KUKA KRL program: CNCRMsgs.src, CNCRMsgs.dat

--- CNCRMsgs.src ---
&ACCESS RV
&REL 50
&PARAM EDITMASK = *
&PARAM TEMPLATE = C:\KRC\Roboter\Template\ExpertVorgabe
DEF CNCRMsgs( )

;************************************************
;              CNC Robotics Ltd
;              www.cncrobotics.co.uk
;************************************************
;     Contact: helpdesk@cncrobotics.co.uk
;     Date: 26/09/23
;     Version: 0.8.51
;************************************************
; Description: message related source files
;************************************************

END

GLOBAL DEF WarningMsg(fin_CNCRMsg:OUT, fin_nGroupNo:IN )

DECL CNCRMessage fin_CNCRMsg
DECL INT fin_nGroupNo

IF fin_CNCRMsg.bDisplayFlag==FALSE THEN

   MsgNotify(fin_CNCRMsg.strMsg[], fin_CNCRMsg.strName[],,,fin_nGroupNo + fin_CNCRMsg.nNo, E_progNotifyMsgOpt)
   fin_CNCRMsg.bDisplayFlag=TRUE
ENDIF

END

GLOBAL DEF DisplayMsg(fin_CNCRMsg:OUT, fin_nGroupNo:IN )

DECL CNCRMessage fin_CNCRMsg
DECL INT fin_nGroupNo

   MsgNotify(fin_CNCRMsg.strMsg[], fin_CNCRMsg.strName[],,,fin_nGroupNo + fin_CNCRMsg.nNo, E_progNotifyMsgOpt)

END

GLOBAL DEF WarningClear(fin_CNCRMsg:OUT )

DECL CNCRMessage fin_CNCRMsg

fin_CNCRMsg.bDisplayFlag= FALSE

END

GLOBAL DEF CheckWarningMsg(bCondition:IN, fin_CNCRMsg:OUT, fin_nGroupNo:IN )

DECL CNCRMessage fin_CNCRMsg
DECL INT fin_nGroupNo
DECL BOOL bCondition

IF bCondition==TRUE THEN
   WarningMsg(fin_CNCRMsg,fin_nGroupNo)
ELSE
   WarningClear(fin_CNCRMsg)

ENDIF

END

GLOBAL DEFFCT INT MessageBoxYesNo(fin_CNCRMsg:OUT, fin_nGroupNo:IN )

DECL CNCRMessage fin_CNCRMsg
DECL INT fin_nGroupNo

DECL INT nAnswer
nAnswer = 0
MsgDialog(nAnswer,fin_CNCRMsg.strMsg[],fin_CNCRMsg.strName[],,,,,,,"No","Yes", FALSE, fin_nGroupNo + fin_CNCRMsg.nNo, E_spsMsgOpt)

return nAnswer

ENDFCT

--- CNCRMsgs.dat ---
&ACCESS  RV
&PARAM DISKPATH = TP/CNCRobotics/Core
&PARAM EDITMASK = *
&PARAM TEMPLATE = C:\KRC\Roboter\Template\ExpertVorgabe
&REL 50
DEFDAT  CNCRMsgs PUBLIC

DECL GLOBAL KRLMSGOPT_T E_progNotifyMsgOpt={VL_STOP FALSE,CLEAR_P_RESET FALSE,LOG_TO_DB TRUE}
DECL GLOBAL KRLMSGOPT_T E_progCommonMsgOpt={VL_STOP TRUE,CLEAR_P_RESET FALSE,LOG_TO_DB TRUE}
DECL GLOBAL KRLMSGOPT_T E_spsMsgOpt={VL_STOP FALSE,CLEAR_P_RESET FALSE,LOG_TO_DB TRUE}

GLOBAL CONST INT nSpsMsg = 0
GLOBAL CONST INT nInterruptMsg = 100
GLOBAL CONST INT nRobotMsg = 200
GLOBAL CONST INT nSpindleMsg = 300
GLOBAL CONST INT nMeasureMsg = 400
GLOBAL CONST INT nToolRackMsg = 500
GLOBAL CONST INT nAutoToolChangeMsg = 600
GLOBAL CONST INT nSystemMsg = 700
GLOBAL CONST INT nMassiveDimensionMsg = 800
GLOBAL CONST INT nFlexxPumpMsg = 900
GLOBAL CONST INT nCEADMsg=1000
GLOBAL CONST INT nSchunkMsg=1400
GLOBAL CONST INT nRoofMsg=1500

GLOBAL STRUC CNCRMessage INT nNo,CHAR strName[24],CHAR strMsg[128],BOOL bDisplayFlag


ENDDAT
